{attribute 'GeneratedUsingTerminal: KL3044-0001'}
{attribute addProperty BoxType "KL3044-0001"}
{attribute addProperty Id "Channel_1AT %I*0Channel_2AT %I*0Channel_3AT %I*0Channel_4AT %I*0"}
{attribute addProperty CRC "2899743849"}
{attribute addProperty Size "0"}
TYPE KL_ACD69469 :
STRUCT
	{attribute addProperty Name "Channel_1"}
	Channel_1 : ;
	{attribute addProperty Name "Channel_2"}
	Channel_2 : ;
	{attribute addProperty Name "Channel_3"}
	Channel_3 : ;
	{attribute addProperty Name "Channel_4"}
	Channel_4 : ;
END_STRUCT
END_TYPE

(* stored: Version 1.2.0.0, ProductVersion 3.1.4024.9
   DUT KL_ACD69469: Id {a0a9625b-3ccc-4fe9-8139-4e2f0eadb372} *)
